# EPICS autosave request: iocBoot/iocEDIO24/auto_settings.req
file "EDIO24_settings.req", P=$(P)
